Staubli VAL3: flushQueue.pgx

public program flushQueue()
  local num l_i
begin
  // This program flushes the queue of object
  //
  // Input param
  //  none
  //
  // Output param
  // none
  //
  // Created 25-09-07                                    C.CURRIVAND
  //----------------------------------------------------------------
  nIdxPush=nIdxPull=0
  for l_i=0 to (nBufferSize-1)
    nEncLatchedVal[l_i]=0
    trDetectedCoord[l_i]=trDEFAULT
    nQueueID[l_i]=nDEFAULTID
    nNumbOfUser[l_i]=0
  endFor
end
